Yaskawa INFORM job: KAROL.JBI

/JOB
//NAME KAROL
//POS
///NPOS 4,4,0,0,0,0
///TOOL 0
///POSTYPE ROBOT
///RECTAN
///RCONF 1,0,0,0,0,0,0,0,0,0,0,0,0,0,0,0,0,0,0,0,0,0,0,0
C00000=1443.693,-296.939,-798.684,-15.7678,-11.8432,-29.6002
///RCONF 0,0,0,0,0,0,0,0,0,0,0,0,0,0,0,0,0,0,0,0,0,0,0,0
C00001=1549.327,232.778,-699.593,37.4202,2.3877,-40.7055
C00002=1549.327,232.778,-699.593,37.4202,2.3877,-40.7055
C00003=1549.326,232.781,-699.593,37.4202,2.3877,-40.7052
BC00000=3693.350
BC00001=3099.006
BC00002=3596.657
BC00003=4355.008
//INST
///DATE 2024/06/19 10:07
///ATTR SC,RW,RJ
////FRAME ROBOT
///GROUP1 RB1,BS1
NOP
MOVJ C00000 BC00000 VJ=50.00
MOVJ C00001 BC00001 VJ=50.00
MOVJ C00002 BC00002 VJ=50.00
MOVJ C00003 BC00003 VJ=50.00
END
